FUNCTION_BLOCK IXP (* Composite FB for boolean input data *)
  (* Standard: 61499-2 *)
  (* Version 1.0, 2024-04-24, franz *)
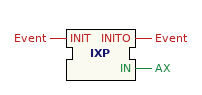
  EVENT_INPUT
    INIT; (* Initialization Request *)
  END_EVENT
  EVENT_OUTPUT
    INITO; (* Initialization Confirm *)
  END_EVENT
  PLUGS
    IN : AX;
  END_PLUGS
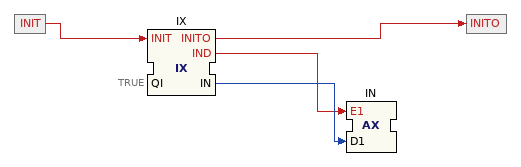
  FBS
    IX : IX(QI := TRUE);
  END_FBS
  EVENT_CONNECTIONS
    INIT TO IX.INIT;
    IX.INITO TO INITO;
    IX.IND TO IN.E1;
  END_CONNECTIONS
  DATA_CONNECTIONS
    IX.IN TO IN.D1;
  END_CONNECTIONS
END_FUNCTION_BLOCK
